{attribute 'GeneratedUsingTerminal: EK1100-0000-0018'}
{attribute addProperty BoxType "EK1100-0000-0018"}
{attribute addProperty Id "Beckhoff_EL25xxEK1122Beckhoff_EL25xxEK1122_6D0E79512A_0001_EL2502_0000_0016EL2502_FF93541015A_0002_EL2502_0000_0017EL2502_FF93541015A_0003_EL2502_0000_0018EL2502_FF93541015A_0004_EL2502_0000_0019EL2502_FF93541015A_0005_EL2502_0000_0020EL2502_FF93541015A_0006_EL2502_0000_0021EL2502_FF93541015A_0007_EL2502_0000_0022EL2502_FF93541015A_0008_EL2502_0000_0023EL2502_FF93541015A_0009_EL2502_0000_0024EL2502_FF93541015A_0010_EL2502_0000_0025EL2502_FF93541015A_0011_EL2502_0000_0026EL2502_FF93541015A_0012_EL2502_0005_0016EL2502_FF93541015A_0013_EL2502_0010_0020EL2502_EABE598A41A_0014_EL2521_0000_0000EL2521_64DF2AB820A_0015_EL2521_0000_1016EL2521_C9F0EF2936A_0016_EL2521_0000_1017EL2521_7FEE0D7136A_0017_EL2521_0000_1018EL2521_7FEE0D7136A_0018_EL2521_0000_1019EL2521_C3BAD9FF36A_0019_EL2521_0000_1020EL2521_C3BAD9FF36A_0020_EL2521_0000_1021EL2521_C3BAD9FF36A_0021_EL2521_0000_1022EL2521_C3BAD9FF36A_0022_EL2521_0024_1016EL2521_64DF2AB820A_0023_EL2521_0024_1017EL2521_64DF2AB820A_0024_EL2521_0024_1018EL2521_C3BAD9FF36A_0025_EL2521_0024_1019EL2521_C3BAD9FF36A_0026_EL2521_0024_1020EL2521_C3BAD9FF36A_0027_EL2521_0024_1021EL2521_C3BAD9FF36A_0028_EL2521_0025_1016EL2521_64DF2AB820A_0029_EL2521_0025_1017EL2521_64DF2AB820A_0030_EL2521_0025_1018EL2521_C3BAD9FF36A_0031_EL2521_0025_1019EL2521_C3BAD9FF36A_0032_EL2521_0025_1020EL2521_C3BAD9FF36A_0033_EL2521_0025_1021EL2521_C3BAD9FF36A_0034_EL2521_0124_0016EL2521_1CEF834B48A_0035_EL2521_0124_0017EL2521_1CEF834B48A_0036_EL2521_0124_0018EL2521_88CAD09450A_0037_EL2521_0124_0019EL2521_88CAD09450A_0038_EL2521_0124_0020EL2521_88CAD09450A_0039_EL2521_1001_0000EL2521_593D4A3218A_0040_EL2521_1001_0001EL2521_64DF2AB820A_0041_EL2521_1001_1016EL2521_64DF2AB820A_0042_EL2521_1001_1017EL2521_64DF2AB820A_0043_EL2521_1001_1018EL2521_C3BAD9FF36A_0044_EL2521_1001_1019EL2521_C3BAD9FF36A_0045_EL2521_1001_1020EL2521_C3BAD9FF36A_0046_EL2522_0000_0017EL2522_8D9DD56772A_0047_EL2522_0000_0018EL2522_8D9DD56772A_0048_EL2522_0000_0021EL2522_8D9DD56772A_0049_EL2522_0000_0022EL2522_8D9DD56772A_0050_EL2535_0000_0016EL2535_27EFEC1532A_0051_EL2535_0000_0017EL2535_27EFEC1532A_0052_EL2535_0000_0018EL2535_27EFEC1532A_0053_EL2535_0000_0019EL2535_27EFEC1532A_0054_EL2535_0000_0021EL2535_27EFEC1532A_0055_EL2535_0000_0022EL2535_27EFEC1532A_0056_EL2535_0000_0023EL2535_27EFEC1532A_0057_EL2535_0002_0016EL2535_27EFEC1532A_0058_EL2535_0002_0017EL2535_27EFEC1532A_0059_EL2535_0002_0018EL2535_27EFEC1532A_0060_EL2535_0002_0019EL2535_27EFEC1532A_0061_EL2535_0002_0020EL2535_27EFEC1532A_0062_EL2535_0002_0021EL2535_27EFEC1532A_0063_EL2535_0002_0022EL2535_27EFEC1532A_0064_EL2535_0002_0023EL2535_27EFEC1532A_0065_EL2535_0005_0022EL2535_27EFEC1532A_0066_EL2535_0005_0023EL2535_27EFEC1532A_0067_EL2535_0050_0016EL2535_27EFEC1532A_0068_EL2535_0050_0017EL2535_27EFEC1532A_0069_EL2535_0050_0018EL2535_27EFEC1532A_0070_EL2535_0050_0019EL2535_27EFEC1532A_0071_EL2535_0050_0020EL2535_27EFEC1532A_0072_EL2535_0050_0021EL2535_27EFEC1532A_0073_EL2535_0050_0022EL2535_27EFEC1532A_0074_EL2535_0050_0023EL2535_27EFEC1532A_0075_EL2535_0100_0019EL2535_27EFEC1532A_0076_EL2535_0100_0020EL2535_27EFEC1532A_0077_EL2535_0100_0021EL2535_27EFEC1532A_0078_EL2535_0100_0022EL2535_27EFEC1532A_0079_EL2535_0100_0023EL2535_27EFEC1532A_0080_EL2535_0103_0023EL2535_CE98521530A_0081_EL2564_0000_0016EL2564_F52874E532A_0082_EL2595_0000_0018EL2595_D2DC76A521A_0083_EL2595_0000_0019EL2595_5796AC7122A_0084_EL2596_0000_0017EL2596_0E9CEA5024A_0085_EL2596_0000_0018EL2596_0E9CEA5024A_0086_EL2596_0010_0016EL2596_0E9CEA5024"}
{attribute addProperty CRC "2416296115"}
{attribute addProperty Size "2720"}
TYPE Beckhoff_EL25xx_9005C0B3 EXTENDS EK1100_AB5A9467 :
STRUCT
	{attribute addProperty Name "Beckhoff_EL25xxEK1122"}
	Beckhoff_EL25xxEK1122 : Beckhoff_EL25xxEK1122_6D0E7951;
	{attribute addProperty Name "A_0001_EL2502_0000_0016"}
	A_0001_EL2502_0000_0016 : EL2502_FF935410;
	{attribute addProperty Name "A_0002_EL2502_0000_0017"}
	A_0002_EL2502_0000_0017 : EL2502_FF935410;
	{attribute addProperty Name "A_0003_EL2502_0000_0018"}
	A_0003_EL2502_0000_0018 : EL2502_FF935410;
	{attribute addProperty Name "A_0004_EL2502_0000_0019"}
	A_0004_EL2502_0000_0019 : EL2502_FF935410;
	{attribute addProperty Name "A_0005_EL2502_0000_0020"}
	A_0005_EL2502_0000_0020 : EL2502_FF935410;
	{attribute addProperty Name "A_0006_EL2502_0000_0021"}
	A_0006_EL2502_0000_0021 : EL2502_FF935410;
	{attribute addProperty Name "A_0007_EL2502_0000_0022"}
	A_0007_EL2502_0000_0022 : EL2502_FF935410;
	{attribute addProperty Name "A_0008_EL2502_0000_0023"}
	A_0008_EL2502_0000_0023 : EL2502_FF935410;
	{attribute addProperty Name "A_0009_EL2502_0000_0024"}
	A_0009_EL2502_0000_0024 : EL2502_FF935410;
	{attribute addProperty Name "A_0010_EL2502_0000_0025"}
	A_0010_EL2502_0000_0025 : EL2502_FF935410;
	{attribute addProperty Name "A_0011_EL2502_0000_0026"}
	A_0011_EL2502_0000_0026 : EL2502_FF935410;
	{attribute addProperty Name "A_0012_EL2502_0005_0016"}
	A_0012_EL2502_0005_0016 : EL2502_FF935410;
	{attribute addProperty Name "A_0013_EL2502_0010_0020"}
	A_0013_EL2502_0010_0020 : EL2502_EABE598A;
	{attribute addProperty Name "A_0014_EL2521_0000_0000"}
	A_0014_EL2521_0000_0000 : EL2521_64DF2AB8;
	{attribute addProperty Name "A_0015_EL2521_0000_1016"}
	A_0015_EL2521_0000_1016 : EL2521_C9F0EF29;
	{attribute addProperty Name "A_0016_EL2521_0000_1017"}
	A_0016_EL2521_0000_1017 : EL2521_7FEE0D71;
	{attribute addProperty Name "A_0017_EL2521_0000_1018"}
	A_0017_EL2521_0000_1018 : EL2521_7FEE0D71;
	{attribute addProperty Name "A_0018_EL2521_0000_1019"}
	A_0018_EL2521_0000_1019 : EL2521_C3BAD9FF;
	{attribute addProperty Name "A_0019_EL2521_0000_1020"}
	A_0019_EL2521_0000_1020 : EL2521_C3BAD9FF;
	{attribute addProperty Name "A_0020_EL2521_0000_1021"}
	A_0020_EL2521_0000_1021 : EL2521_C3BAD9FF;
	{attribute addProperty Name "A_0021_EL2521_0000_1022"}
	A_0021_EL2521_0000_1022 : EL2521_C3BAD9FF;
	{attribute addProperty Name "A_0022_EL2521_0024_1016"}
	A_0022_EL2521_0024_1016 : EL2521_64DF2AB8;
	{attribute addProperty Name "A_0023_EL2521_0024_1017"}
	A_0023_EL2521_0024_1017 : EL2521_64DF2AB8;
	{attribute addProperty Name "A_0024_EL2521_0024_1018"}
	A_0024_EL2521_0024_1018 : EL2521_C3BAD9FF;
	{attribute addProperty Name "A_0025_EL2521_0024_1019"}
	A_0025_EL2521_0024_1019 : EL2521_C3BAD9FF;
	{attribute addProperty Name "A_0026_EL2521_0024_1020"}
	A_0026_EL2521_0024_1020 : EL2521_C3BAD9FF;
	{attribute addProperty Name "A_0027_EL2521_0024_1021"}
	A_0027_EL2521_0024_1021 : EL2521_C3BAD9FF;
	{attribute addProperty Name "A_0028_EL2521_0025_1016"}
	A_0028_EL2521_0025_1016 : EL2521_64DF2AB8;
	{attribute addProperty Name "A_0029_EL2521_0025_1017"}
	A_0029_EL2521_0025_1017 : EL2521_64DF2AB8;
	{attribute addProperty Name "A_0030_EL2521_0025_1018"}
	A_0030_EL2521_0025_1018 : EL2521_C3BAD9FF;
	{attribute addProperty Name "A_0031_EL2521_0025_1019"}
	A_0031_EL2521_0025_1019 : EL2521_C3BAD9FF;
	{attribute addProperty Name "A_0032_EL2521_0025_1020"}
	A_0032_EL2521_0025_1020 : EL2521_C3BAD9FF;
	{attribute addProperty Name "A_0033_EL2521_0025_1021"}
	A_0033_EL2521_0025_1021 : EL2521_C3BAD9FF;
	{attribute addProperty Name "A_0034_EL2521_0124_0016"}
	A_0034_EL2521_0124_0016 : EL2521_1CEF834B;
	{attribute addProperty Name "A_0035_EL2521_0124_0017"}
	A_0035_EL2521_0124_0017 : EL2521_1CEF834B;
	{attribute addProperty Name "A_0036_EL2521_0124_0018"}
	A_0036_EL2521_0124_0018 : EL2521_88CAD094;
	{attribute addProperty Name "A_0037_EL2521_0124_0019"}
	A_0037_EL2521_0124_0019 : EL2521_88CAD094;
	{attribute addProperty Name "A_0038_EL2521_0124_0020"}
	A_0038_EL2521_0124_0020 : EL2521_88CAD094;
	{attribute addProperty Name "A_0039_EL2521_1001_0000"}
	A_0039_EL2521_1001_0000 : EL2521_593D4A32;
	{attribute addProperty Name "A_0040_EL2521_1001_0001"}
	A_0040_EL2521_1001_0001 : EL2521_64DF2AB8;
	{attribute addProperty Name "A_0041_EL2521_1001_1016"}
	A_0041_EL2521_1001_1016 : EL2521_64DF2AB8;
	{attribute addProperty Name "A_0042_EL2521_1001_1017"}
	A_0042_EL2521_1001_1017 : EL2521_64DF2AB8;
	{attribute addProperty Name "A_0043_EL2521_1001_1018"}
	A_0043_EL2521_1001_1018 : EL2521_C3BAD9FF;
	{attribute addProperty Name "A_0044_EL2521_1001_1019"}
	A_0044_EL2521_1001_1019 : EL2521_C3BAD9FF;
	{attribute addProperty Name "A_0045_EL2521_1001_1020"}
	A_0045_EL2521_1001_1020 : EL2521_C3BAD9FF;
	{attribute addProperty Name "A_0046_EL2522_0000_0017"}
	A_0046_EL2522_0000_0017 : EL2522_8D9DD567;
	{attribute addProperty Name "A_0047_EL2522_0000_0018"}
	A_0047_EL2522_0000_0018 : EL2522_8D9DD567;
	{attribute addProperty Name "A_0048_EL2522_0000_0021"}
	A_0048_EL2522_0000_0021 : EL2522_8D9DD567;
	{attribute addProperty Name "A_0049_EL2522_0000_0022"}
	A_0049_EL2522_0000_0022 : EL2522_8D9DD567;
	{attribute addProperty Name "A_0050_EL2535_0000_0016"}
	A_0050_EL2535_0000_0016 : EL2535_27EFEC15;
	{attribute addProperty Name "A_0051_EL2535_0000_0017"}
	A_0051_EL2535_0000_0017 : EL2535_27EFEC15;
	{attribute addProperty Name "A_0052_EL2535_0000_0018"}
	A_0052_EL2535_0000_0018 : EL2535_27EFEC15;
	{attribute addProperty Name "A_0053_EL2535_0000_0019"}
	A_0053_EL2535_0000_0019 : EL2535_27EFEC15;
	{attribute addProperty Name "A_0054_EL2535_0000_0021"}
	A_0054_EL2535_0000_0021 : EL2535_27EFEC15;
	{attribute addProperty Name "A_0055_EL2535_0000_0022"}
	A_0055_EL2535_0000_0022 : EL2535_27EFEC15;
	{attribute addProperty Name "A_0056_EL2535_0000_0023"}
	A_0056_EL2535_0000_0023 : EL2535_27EFEC15;
	{attribute addProperty Name "A_0057_EL2535_0002_0016"}
	A_0057_EL2535_0002_0016 : EL2535_27EFEC15;
	{attribute addProperty Name "A_0058_EL2535_0002_0017"}
	A_0058_EL2535_0002_0017 : EL2535_27EFEC15;
	{attribute addProperty Name "A_0059_EL2535_0002_0018"}
	A_0059_EL2535_0002_0018 : EL2535_27EFEC15;
	{attribute addProperty Name "A_0060_EL2535_0002_0019"}
	A_0060_EL2535_0002_0019 : EL2535_27EFEC15;
	{attribute addProperty Name "A_0061_EL2535_0002_0020"}
	A_0061_EL2535_0002_0020 : EL2535_27EFEC15;
	{attribute addProperty Name "A_0062_EL2535_0002_0021"}
	A_0062_EL2535_0002_0021 : EL2535_27EFEC15;
	{attribute addProperty Name "A_0063_EL2535_0002_0022"}
	A_0063_EL2535_0002_0022 : EL2535_27EFEC15;
	{attribute addProperty Name "A_0064_EL2535_0002_0023"}
	A_0064_EL2535_0002_0023 : EL2535_27EFEC15;
	{attribute addProperty Name "A_0065_EL2535_0005_0022"}
	A_0065_EL2535_0005_0022 : EL2535_27EFEC15;
	{attribute addProperty Name "A_0066_EL2535_0005_0023"}
	A_0066_EL2535_0005_0023 : EL2535_27EFEC15;
	{attribute addProperty Name "A_0067_EL2535_0050_0016"}
	A_0067_EL2535_0050_0016 : EL2535_27EFEC15;
	{attribute addProperty Name "A_0068_EL2535_0050_0017"}
	A_0068_EL2535_0050_0017 : EL2535_27EFEC15;
	{attribute addProperty Name "A_0069_EL2535_0050_0018"}
	A_0069_EL2535_0050_0018 : EL2535_27EFEC15;
	{attribute addProperty Name "A_0070_EL2535_0050_0019"}
	A_0070_EL2535_0050_0019 : EL2535_27EFEC15;
	{attribute addProperty Name "A_0071_EL2535_0050_0020"}
	A_0071_EL2535_0050_0020 : EL2535_27EFEC15;
	{attribute addProperty Name "A_0072_EL2535_0050_0021"}
	A_0072_EL2535_0050_0021 : EL2535_27EFEC15;
	{attribute addProperty Name "A_0073_EL2535_0050_0022"}
	A_0073_EL2535_0050_0022 : EL2535_27EFEC15;
	{attribute addProperty Name "A_0074_EL2535_0050_0023"}
	A_0074_EL2535_0050_0023 : EL2535_27EFEC15;
	{attribute addProperty Name "A_0075_EL2535_0100_0019"}
	A_0075_EL2535_0100_0019 : EL2535_27EFEC15;
	{attribute addProperty Name "A_0076_EL2535_0100_0020"}
	A_0076_EL2535_0100_0020 : EL2535_27EFEC15;
	{attribute addProperty Name "A_0077_EL2535_0100_0021"}
	A_0077_EL2535_0100_0021 : EL2535_27EFEC15;
	{attribute addProperty Name "A_0078_EL2535_0100_0022"}
	A_0078_EL2535_0100_0022 : EL2535_27EFEC15;
	{attribute addProperty Name "A_0079_EL2535_0100_0023"}
	A_0079_EL2535_0100_0023 : EL2535_27EFEC15;
	{attribute addProperty Name "A_0080_EL2535_0103_0023"}
	A_0080_EL2535_0103_0023 : EL2535_CE985215;
	{attribute addProperty Name "A_0081_EL2564_0000_0016"}
	A_0081_EL2564_0000_0016 : EL2564_F52874E5;
	{attribute addProperty Name "A_0082_EL2595_0000_0018"}
	A_0082_EL2595_0000_0018 : EL2595_D2DC76A5;
	{attribute addProperty Name "A_0083_EL2595_0000_0019"}
	A_0083_EL2595_0000_0019 : EL2595_5796AC71;
	{attribute addProperty Name "A_0084_EL2596_0000_0017"}
	A_0084_EL2596_0000_0017 : EL2596_0E9CEA50;
	{attribute addProperty Name "A_0085_EL2596_0000_0018"}
	A_0085_EL2596_0000_0018 : EL2596_0E9CEA50;
	{attribute addProperty Name "A_0086_EL2596_0010_0016"}
	A_0086_EL2596_0010_0016 : EL2596_0E9CEA50;
END_STRUCT
END_TYPE

(* stored: Version 1.2.0.0, ProductVersion 3.1.4024.9
   DUT Beckhoff_EL25xx_9005C0B3: Id {e90bf5be-ca97-4068-878f-a37df4f57470} *)
